PROGRAM MAIN
VAR
	Machine : FB_Machine;
END_VAR

PRG_LoadTwinSAFE();
Machine();

END_PROGRAM

(* stored: Version 1.1.0.1, ProductVersion 3.1.4024.13
   POU MAIN: Id {aa01f370-733e-448c-acf5-951e36636772}, SpecialFunc None *)
